FUNCTION_BLOCK WPMaster (* Basic Function Block Type *)
  (* Standard: 61499-2 *)
  (* Version 0.2, 2003-12-04, JHC, Rockwell Automation, Renamed for better indexing. *)
  (* Version 0.1, 2002-11-05, JHC, Rockwell Automation, Corrected missing ST element in Algorithm REQ. *)
  (* Version 0.0, 2000-05-30, JHC, Rockwell Automation *)
  (* Compiler header: package fb.rt.pnp; *)
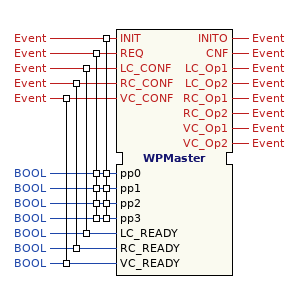
  EVENT_INPUT
    INIT WITH pp0, pp1, pp2, pp3; (* Initialization Request *)
    REQ WITH pp0, pp1, pp2, pp3; (* Normal Execution Request *)
    LC_CONF WITH LC_READY;
    RC_CONF WITH RC_READY;
    VC_CONF WITH VC_READY;
  END_EVENT
  EVENT_OUTPUT
    INITO; (* Initialization Confirm *)
    CNF; (* Execution Confirmation *)
    LC_Op1;
    LC_Op2;
    RC_Op1;
    RC_Op2;
    VC_Op1;
    VC_Op2;
  END_EVENT
  VAR_INPUT
    pp0 : BOOL;
    pp1 : BOOL;
    pp2 : BOOL;
    pp3 : BOOL;
    LC_READY : BOOL;
    RC_READY : BOOL;
    VC_READY : BOOL;
  END_VAR
  VAR
    Flag : BOOL;
  END_VAR
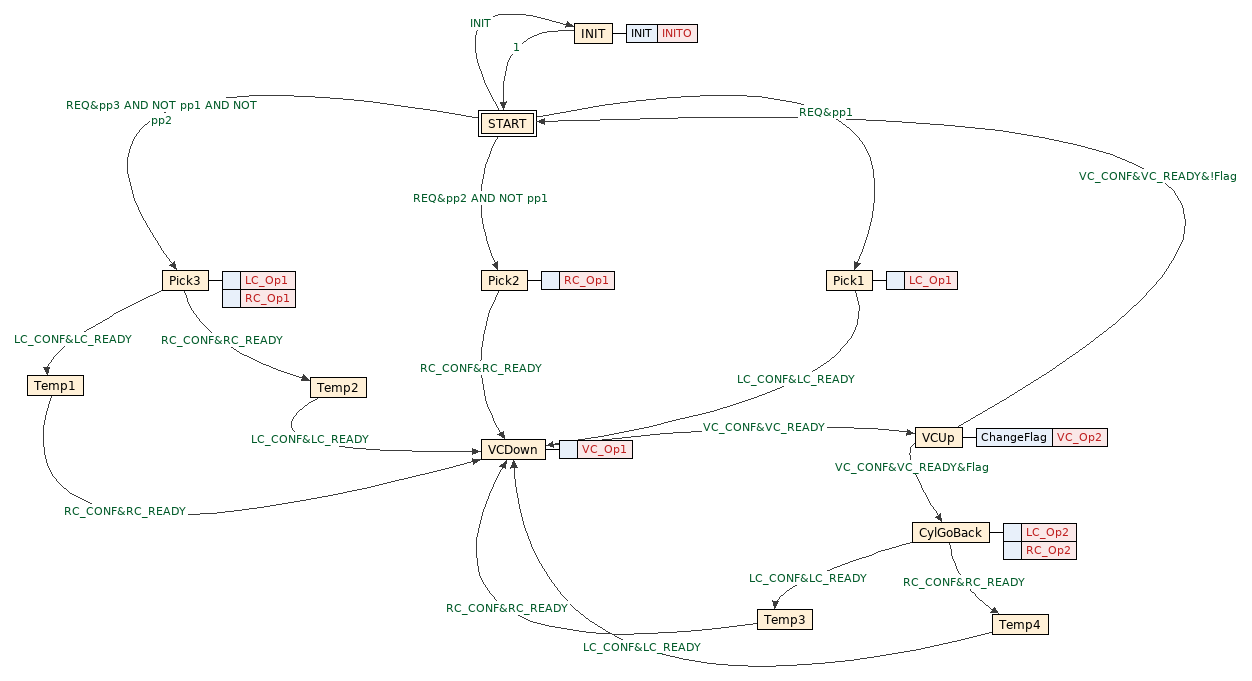
  EC_STATES
    START; (* Initial State *)
    INIT : INIT -> INITO; (* Initialization *)
    Pick1 : -> LC_Op1;
    Pick2 : -> RC_Op1;
    Pick3 : -> LC_Op1, -> RC_Op1;
    VCDown : -> VC_Op1;
    VCUp : ChangeFlag -> VC_Op2;
    CylGoBack : -> LC_Op2, -> RC_Op2;
    Temp1;
    Temp2;
    Temp3;
    Temp4;
  END_STATES
  EC_TRANSITIONS
    START TO INIT := INIT;
    INIT TO START := 1;
    START TO Pick1 := REQ&pp1;
    START TO Pick2 := REQ&pp2 AND NOT pp1;
    START TO Pick3 := REQ&pp3 AND NOT pp1 AND NOT  pp2;
    Pick1 TO VCDown := LC_CONF&LC_READY;
    Pick2 TO VCDown := RC_CONF&RC_READY;
    VCDown TO VCUp := VC_CONF&VC_READY;
    VCUp TO CylGoBack := VC_CONF&VC_READY&Flag;
    Pick3 TO Temp1 := LC_CONF&LC_READY;
    Pick3 TO Temp2 := RC_CONF&RC_READY;
    Temp2 TO VCDown := LC_CONF&LC_READY;
    Temp1 TO VCDown := RC_CONF&RC_READY;
    CylGoBack TO Temp3 := LC_CONF&LC_READY;
    CylGoBack TO Temp4 := RC_CONF&RC_READY;
    Temp3 TO VCDown := RC_CONF&RC_READY;
    Temp4 TO VCDown := LC_CONF&LC_READY;
    VCUp TO START := VC_CONF&VC_READY&!Flag;
  END_TRANSITIONS
  ALGORITHM INIT IN ST: (* Initialization algorithm *)
Flag := FALSE;
  END_ALGORITHM
  ALGORITHM REQ IN ST: (* Normally executed algorithm *)

  END_ALGORITHM
  ALGORITHM ChangeFlag IN ST:
if Flag THEN
Flag := FALSE;
ELSE
Flag := TRUE;
END_IF

System.out.println("ChangeFlag!!"+Flag);
  END_ALGORITHM
END_FUNCTION_BLOCK
